{attribute addProperty BoxType "EK1100-0000-0018"}
{attribute addProperty Id "Beckhoff_EJ2xxxEK1122Beckhoff_EJ2xxxEK1122_7BCCD4D9162A_0001_EJ2008_0000_0017EJ2008_A854BE6D8110.125A_0002_EJ2008_0000_0018EJ2008_A854BE6D8110.125A_0003_EJ2128_0000_0016EJ2128_A854BE6D8110.125A_0004_EJ2502_0000_0023EJ2502_68F74D5A11314.125A_0005_EJ2502_0000_0024EJ2502_68F74D5A11314.125A_0006_EJ2521_0224_0016EJ2521_A10F5EEB35444.25A_0007_EJ2522_0000_0022EJ2522_58A1BC1F43454.25A_0008_EJ2809_0000_0017EJ2809_859F43D214518.125A_0009_EJ2889_0000_0016EJ2889_859F43D214518.125A_0010_EJ2889_0000_0017EJ2889_859F43D214518.125"}
{attribute addProperty CRC "1123332187"}
{attribute addProperty SizeInBites "1708"}
{attribute addProperty SizeInBytes "213.5"}
TYPE Beckhoff_EJ2xxx_42F4B05B EXTENDS EK1100_179A0949 :
STRUCT
	{attribute addProperty Name "Beckhoff_EJ2xxxEK1122"}
	Beckhoff_EJ2xxxEK1122 : Beckhoff_EJ2xxxEK1122_7BCCD4D9;
	{attribute addProperty Name "A_0001_EJ2008_0000_0017"}
	A_0001_EJ2008_0000_0017 : EJ2008_A854BE6D;
	{attribute addProperty Name "A_0002_EJ2008_0000_0018"}
	A_0002_EJ2008_0000_0018 : EJ2008_A854BE6D;
	{attribute addProperty Name "A_0003_EJ2128_0000_0016"}
	A_0003_EJ2128_0000_0016 : EJ2128_A854BE6D;
	{attribute addProperty Name "A_0004_EJ2502_0000_0023"}
	A_0004_EJ2502_0000_0023 : EJ2502_68F74D5A;
	{attribute addProperty Name "A_0005_EJ2502_0000_0024"}
	A_0005_EJ2502_0000_0024 : EJ2502_68F74D5A;
	{attribute addProperty Name "A_0006_EJ2521_0224_0016"}
	A_0006_EJ2521_0224_0016 : EJ2521_A10F5EEB;
	{attribute addProperty Name "A_0007_EJ2522_0000_0022"}
	A_0007_EJ2522_0000_0022 : EJ2522_58A1BC1F;
	{attribute addProperty Name "A_0008_EJ2809_0000_0017"}
	A_0008_EJ2809_0000_0017 : EJ2809_859F43D2;
	{attribute addProperty Name "A_0009_EJ2889_0000_0016"}
	A_0009_EJ2889_0000_0016 : EJ2889_859F43D2;
	{attribute addProperty Name "A_0010_EJ2889_0000_0017"}
	A_0010_EJ2889_0000_0017 : EJ2889_859F43D2;
END_STRUCT
END_TYPE

(* stored: Version 1.2.0.0, ProductVersion 3.1.4024.9
   DUT Beckhoff_EJ2xxx_42F4B05B: Id {e184580c-3ecf-4b2a-8745-8ba91d568e29} *)
